Staubli VAL3: getdWordAt.pgx

public program getDwordAt(num x_nByteIndex, num& x_nBuffer[], num& x_nRes)
begin

  //Header begin

  //This function return in "x_nRes" the value of the double word composed by four bytes starting from "x_nByteIndex" element of the array x_nBuffer (most likely a plc's memory area you read with readArea()).
  //The first byte is the lower part of the word (Big Endian)
  //
  //Input parameters
  //
  //num x_nByteIndex: the index of the element in the "x_nBuffer[]" array representing the starting byte of the double word we want to read
	//num x_nBuffer[1]: the monodimensional array of num from where we are reading a double word.
  //
  //Output parameters
  //
  // num x_nRes: where the result is stored.
  //
  //Examples
  //
  // 	call getDWordAt(7, nDB, l_nRes)
  //
  //History
  // Creation: 24-12-16 - Alessio Villa
  //Header end

  x_nRes=x_nBuffer[x_nByteIndex]*power(2,24)+x_nBuffer[x_nByteIndex+1]*power(2,16)+x_nBuffer[x_nByteIndex+2]*power(2,8)+x_nBuffer[x_nByteIndex+3]

end
